{attribute 'qualified_only'}
{attribute 'strict'}
TYPE E_FCU_ControlMode :
(
	Position := 0,
	Force := 1,
	SoftTouch := 3
) WORD;
END_TYPE

(* stored: Version 1.1.0.1, ProductVersion 3.1.4024.9
   DUT E_FCU_ControlMode: Id {f252bdbd-98f8-4319-bb1a-ebd9a05a3666} *)
